{attribute 'qualified_only'}
VAR_GLOBAL
	mb_Input_Coils    	:	ARRAY [0..511] OF BOOL;
	mb_Output_Coils 	:   ARRAY [0..511] OF BOOL;
 	mb_Input_Registers 	:   ARRAY [0..511] OF WORD;
 	mb_Output_Registers :   ARRAY [0..255] OF WORD;
	
	nInputCoilIndex: INT;
	nOutputCoilIndex: INT;
	nInputRegisterIndex: INT;
	nOutputRegisterIndex: INT;
END_VAR

(* stored: Version 1.1.0.1, ProductVersion 3.1.4024.12
   GVL GVL: Id {ec8d8fc1-a1fb-4ef2-9bc9-97beb9d6cc69} *)
